(* IEC 61131-3 sources: horner-cscape-mcp/artifacts/projects/TankLevelClosedLoop/pous, 5 files *)

(* ---- AlarmMonitor.st ---- *)
PROGRAM AlarmMonitor
VAR trip : BOOL; END_VAR
trip := FALSE;
END_PROGRAM

(* ---- AuxPumpControl.st ---- *)
PROGRAM AuxPumpControl
VAR cmd : BOOL; END_VAR
cmd := TRUE;
END_PROGRAM

(* ---- BrokenPOU.st ---- *)
PROGRAM BrokenPOU
VAR
    RawVal : INT;
END_VAR

RawVal := 10 + 5;
END_PROGRAM

(* ---- SafetyInterlockST.st ---- *)
PROGRAM SafetyInterlockST
VAR x : INT; END_VAR
x := 1;
END_PROGRAM

(* ---- TankLevelClosedLoop.st ---- *)
PROGRAM TankLevelClosedLoop
VAR
    Setpoint : REAL := 60.0;
    TankLevelPV : REAL := 50.0;
    Error : REAL := 0.0;
    ControlOutput : REAL := 0.0;
    Kp : REAL := 2.5;
END_VAR

(* Simple Tank-Level Closed Loop: Setpoint, Measured Level, Error, Output *)
Error := Setpoint - TankLevelPV;
ControlOutput := Kp * Error;

IF ControlOutput > 100.0 THEN
    ControlOutput := 100.0;
ELSIF ControlOutput < 0.0 THEN
    ControlOutput := 0.0;
END_IF;
END_PROGRAM
